SUBAPPLICATION mapping_Uebung_017 (* Control Audio Signal *)
  (* Standard: 61499-2 *)
  (* Version 1.0, 2023-10-23, franz *)
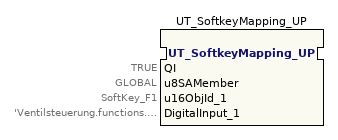
  FBS
    UT_SoftkeyMapping_UP : UT_SoftkeyMapping_UP(QI := TRUE, u8SAMember := GLOBAL, u16ObjId_1 := SoftKey_F1, DigitalInput_1 := 'Ventilsteuerung.functions.SoftKey_F1_UP');
  END_FBS
END_SUBAPPLICATION
